Staubli VAL3: sockets.pjx

Parameters version=s7.2 stackSize=0 millimeterUnit=true
Data file=sockets.dtx
